{attribute 'qualified_only'}
{attribute 'strict'}
TYPE E_StepAxle :
(
	//Idle	        := 0,
  Init          := 1,
  
	// STEPS ABSOLUTE
 	MoveAbs		    := 11,
	EndMoveAbs    := 12,
  
	// STEPS STOP
  InitStop      := 50,
	Stopping		  := 51,
  EndStopping   := 52,
	
	// STEPS HOMING
  InitHoming    := 60,
	Homing			  := 61,
  EndHoming     := 62,
  InitAbortHoming := 63,
  AbortHoming   := 64,
  InitRetryHoming := 65,
  RetryHoming     := 66,
	
	// STEPS Reset
  ResetTimeout := 70,
	Resetting	:= 71,
  ResetEnd := 72,
  
  // step jogs
  JogMoveFW := 80,
  JogMoveBW := 81,
  JogStop := 82,
  JogEnd := 83
);
END_TYPE

(* stored: Version 1.1.0.1, ProductVersion 3.1.4024.12
   DUT E_StepAxle: Id {9d1461ca-9455-4ec7-9499-14ba825dea07} *)
